KUKA KRL program: tool_gut_s.src, tool_gut_s.dat

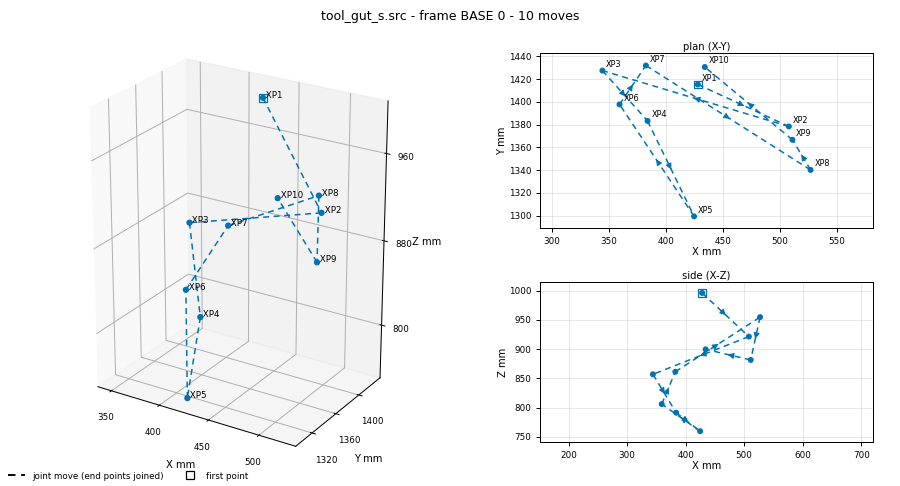
[picture p0: tool path of tool_gut_s.src in frame BASE 0, 10 of 12 moves have a stored position in this frame; points joined in program order, loops and branches not executed]
--- tool_gut_s.src ---
&ACCESS RVO
&REL 1
&PARAM EDITMASK = *
&PARAM TEMPLATE = C:\KRC\Roboter\Template\vorgabe
DEF tool_gut_s( )
;FOLD INI;%{PE}
  ;FOLD BASISTECH INI
    GLOBAL INTERRUPT DECL 3 WHEN $STOPMESS==TRUE DO IR_STOPM ( )
    INTERRUPT ON 3
    BAS (#INITMOV,0 )
  ;ENDFOLD (BASISTECH INI)
  ;FOLD USER INI
    ;Make your modifications here

  ;ENDFOLD (USER INI)
;ENDFOLD (INI)

;FOLD PTP HOME Vel=10 % DEFAULT;%{PE}%R 8.3.40,%MKUKATPBASIS,%CMOVE,%VPTP,%P 1:PTP, 2:HOME, 3:, 5:10, 7:DEFAULT
$BWDSTART=FALSE
PDAT_ACT=PDEFAULT
FDAT_ACT=FHOME
BAS(#PTP_PARAMS,10)
$H_POS=XHOME
PTP XHOME
;ENDFOLD

WAIT FOR IS_KEY_PRESSED(12)

;FOLD PTP P1 Vel=30 % PDAT1 Tool[11]:jan_ba Base[0];%{PE}%R 8.3.40,%MKUKATPBASIS,%CMOVE,%VPTP,%P 1:PTP, 2:P1, 3:, 5:30, 7:PDAT1
$BWDSTART=FALSE
PDAT_ACT=PPDAT1
FDAT_ACT=FP1
BAS(#PTP_PARAMS,30)
PTP XP1
;ENDFOLD

WAIT FOR IS_KEY_PRESSED(12)

;FOLD PTP P2 Vel=30 % PDAT2 Tool[11]:jan_ba Base[0];%{PE}%R 8.3.40,%MKUKATPBASIS,%CMOVE,%VPTP,%P 1:PTP, 2:P2, 3:, 5:30, 7:PDAT2
$BWDSTART=FALSE
PDAT_ACT=PPDAT2
FDAT_ACT=FP2
BAS(#PTP_PARAMS,30)
PTP XP2
;ENDFOLD

WAIT FOR IS_KEY_PRESSED(12)

;FOLD PTP P3 Vel=30 % PDAT3 Tool[11]:jan_ba Base[0];%{PE}%R 8.3.40,%MKUKATPBASIS,%CMOVE,%VPTP,%P 1:PTP, 2:P3, 3:, 5:30, 7:PDAT3
$BWDSTART=FALSE
PDAT_ACT=PPDAT3
FDAT_ACT=FP3
BAS(#PTP_PARAMS,30)
PTP XP3
;ENDFOLD

WAIT FOR IS_KEY_PRESSED(12)

;FOLD PTP P4 Vel=30 % PDAT4 Tool[11]:jan_ba Base[0];%{PE}%R 8.3.40,%MKUKATPBASIS,%CMOVE,%VPTP,%P 1:PTP, 2:P4, 3:, 5:30, 7:PDAT4
$BWDSTART=FALSE
PDAT_ACT=PPDAT4
FDAT_ACT=FP4
BAS(#PTP_PARAMS,30)
PTP XP4
;ENDFOLD

WAIT FOR IS_KEY_PRESSED(12)


;FOLD PTP P5 Vel=30 % PDAT5 Tool[11]:jan_ba Base[0];%{PE}%R 8.3.40,%MKUKATPBASIS,%CMOVE,%VPTP,%P 1:PTP, 2:P5, 3:, 5:30, 7:PDAT5
$BWDSTART=FALSE
PDAT_ACT=PPDAT5
FDAT_ACT=FP5
BAS(#PTP_PARAMS,30)
PTP XP5
;ENDFOLD

WAIT FOR IS_KEY_PRESSED(12)

;FOLD PTP P6 Vel=30 % PDAT6 Tool[11]:jan_ba Base[0];%{PE}%R 8.3.40,%MKUKATPBASIS,%CMOVE,%VPTP,%P 1:PTP, 2:P6, 3:, 5:30, 7:PDAT6
$BWDSTART=FALSE
PDAT_ACT=PPDAT6
FDAT_ACT=FP6
BAS(#PTP_PARAMS,30)
PTP XP6
;ENDFOLD

WAIT FOR IS_KEY_PRESSED(12)

;FOLD PTP P7 Vel=30 % PDAT7 Tool[11]:jan_ba Base[0];%{PE}%R 8.3.40,%MKUKATPBASIS,%CMOVE,%VPTP,%P 1:PTP, 2:P7, 3:, 5:30, 7:PDAT7
$BWDSTART=FALSE
PDAT_ACT=PPDAT7
FDAT_ACT=FP7
BAS(#PTP_PARAMS,30)
PTP XP7
;ENDFOLD

WAIT FOR IS_KEY_PRESSED(12)

;FOLD PTP P8 Vel=30 % PDAT8 Tool[11]:jan_ba Base[0];%{PE}%R 8.3.40,%MKUKATPBASIS,%CMOVE,%VPTP,%P 1:PTP, 2:P8, 3:, 5:30, 7:PDAT8
$BWDSTART=FALSE
PDAT_ACT=PPDAT8
FDAT_ACT=FP8
BAS(#PTP_PARAMS,30)
PTP XP8
;ENDFOLD

WAIT FOR IS_KEY_PRESSED(12)

;FOLD PTP P9 Vel=30 % PDAT9 Tool[11]:jan_ba Base[0];%{PE}%R 8.3.40,%MKUKATPBASIS,%CMOVE,%VPTP,%P 1:PTP, 2:P9, 3:, 5:30, 7:PDAT9
$BWDSTART=FALSE
PDAT_ACT=PPDAT9
FDAT_ACT=FP9
BAS(#PTP_PARAMS,30)
PTP XP9
;ENDFOLD

WAIT FOR IS_KEY_PRESSED(12)

;FOLD PTP P10 Vel=30 % PDAT10 Tool[11]:jan_ba Base[0];%{PE}%R 8.3.40,%MKUKATPBASIS,%CMOVE,%VPTP,%P 1:PTP, 2:P10, 3:, 5:30, 7:PDAT10
$BWDSTART=FALSE
PDAT_ACT=PPDAT10
FDAT_ACT=FP10
BAS(#PTP_PARAMS,30)
PTP XP10
;ENDFOLD


WAIT FOR IS_KEY_PRESSED(12)



;FOLD PTP HOME Vel=10 % DEFAULT;%{PE}%R 8.3.40,%MKUKATPBASIS,%CMOVE,%VPTP,%P 1:PTP, 2:HOME, 3:, 5:10, 7:DEFAULT
$BWDSTART=FALSE
PDAT_ACT=PDEFAULT
FDAT_ACT=FHOME
BAS(#PTP_PARAMS,10)
$H_POS=XHOME
PTP XHOME
;ENDFOLD

END

--- tool_gut_s.dat ---
&ACCESS RVO
&REL 1
&PARAM EDITMASK = *
&PARAM TEMPLATE = C:\KRC\Roboter\Template\vorgabe
DEFDAT  tool_gut_s
;FOLD EXTERNAL DECLARATIONS;%{PE}%MKUKATPBASIS,%CEXT,%VCOMMON,%P
;FOLD BASISTECH EXT;%{PE}%MKUKATPBASIS,%CEXT,%VEXT,%P
EXT  BAS (BAS_COMMAND  :IN,REAL  :IN )
DECL INT SUCCESS
;ENDFOLD (BASISTECH EXT)
;FOLD USER EXT;%{E}%MKUKATPUSER,%CEXT,%VEXT,%P
;Make your modifications here

;ENDFOLD (USER EXT)
;ENDFOLD (EXTERNAL DECLARATIONS)
DECL BASIS_SUGG_T LAST_BASIS={POINT1[] "P10                     ",POINT2[] "P10                     ",CP_PARAMS[] "CPDAT0                  ",PTP_PARAMS[] "PDAT10                  ",CONT[] "                        ",CP_VEL[] "2.0                     ",PTP_VEL[] "30                      ",SYNC_PARAMS[] "SYNCDAT                 ",SPL_NAME[] "S0                      ",A_PARAMS[] "ADAT0                   "}
DECL E6POS XP1={X 428.073151,Y 1415.33362,Z 995.893921,A 45.0438805,B 61.3839645,C -21.8034782,S 22,T 27,E1 0.00486961612,E2 20159.9980,E3 0.0,E4 0.0,E5 0.0,E6 0.0}
DECL FDAT FP1={TOOL_NO 11,BASE_NO 0,IPO_FRAME #BASE,POINT2[] " ",TQ_STATE FALSE}
DECL PDAT PPDAT1={VEL 100.000,ACC 50.0000,APO_DIST 100.000,APO_MODE #CDIS,GEAR_JERK 50.0000,EXAX_IGN 0}
DECL E6POS XP2={X 508.024689,Y 1378.40088,Z 921.330078,A -49.0426292,B 81.0973740,C -87.4984,S 22,T 27,E1 0.00486961100,E2 20159.9980,E3 0.0,E4 0.0,E5 0.0,E6 0.0}
DECL FDAT FP2={TOOL_NO 11,BASE_NO 0,IPO_FRAME #BASE,POINT2[] " ",TQ_STATE FALSE}
DECL PDAT PPDAT2={VEL 100.000,ACC 50.0000,APO_DIST 100.000,APO_MODE #CDIS,GEAR_JERK 50.0000,EXAX_IGN 0}
DECL E6POS XP3={X 344.155914,Y 1427.50085,Z 856.935913,A -65.5491104,B 67.6447372,C -167.687149,S 22,T 51,E1 0.00486961612,E2 20159.9980,E3 0.0,E4 0.0,E5 0.0,E6 0.0}
DECL FDAT FP3={TOOL_NO 11,BASE_NO 0,IPO_FRAME #BASE,POINT2[] " ",TQ_STATE FALSE}
DECL PDAT PPDAT3={VEL 100.000,ACC 50.0000,APO_DIST 100.000,APO_MODE #CDIS,GEAR_JERK 50.0000,EXAX_IGN 0}
DECL E6POS XP4={X 383.834961,Y 1383.27515,Z 791.314087,A -25.8400383,B 17.3074379,C -142.470688,S 22,T 19,E1 0.00486961612,E2 20159.9980,E3 0.0,E4 0.0,E5 0.0,E6 0.0}
DECL FDAT FP4={TOOL_NO 11,BASE_NO 0,IPO_FRAME #BASE,POINT2[] " ",TQ_STATE FALSE}
DECL PDAT PPDAT4={VEL 100.000,ACC 50.0000,APO_DIST 100.000,APO_MODE #CDIS,GEAR_JERK 50.0000,EXAX_IGN 0}
DECL E6POS XP5={X 424.737366,Y 1299.38477,Z 759.745,A -47.7535095,B -4.85419083,C -161.114349,S 18,T 3,E1 0.00486961612,E2 20159.9980,E3 0.0,E4 0.0,E5 0.0,E6 0.0}
DECL FDAT FP5={TOOL_NO 11,BASE_NO 0,IPO_FRAME #BASE,POINT2[] " ",TQ_STATE FALSE}
DECL PDAT PPDAT5={VEL 100.000,ACC 50.0000,APO_DIST 100.000,APO_MODE #CDIS,GEAR_JERK 50.0000,EXAX_IGN 0}
DECL E6POS XP6={X 359.204346,Y 1397.80554,Z 806.092102,A -4.80768585,B 12.8503466,C -133.435959,S 22,T 19,E1 0.00486961612,E2 20159.9980,E3 0.0,E4 0.0,E5 0.0,E6 0.0}
DECL FDAT FP6={TOOL_NO 11,BASE_NO 0,IPO_FRAME #BASE,POINT2[] " ",TQ_STATE FALSE}
DECL PDAT PPDAT6={VEL 100.000,ACC 50.0000,APO_DIST 100.000,APO_MODE #CDIS,GEAR_JERK 50.0000,EXAX_IGN 0}
DECL E6POS XP7={X 382.381470,Y 1431.97205,Z 861.245178,A -1.15962076,B -4.24653769,C -110.314613,S 22,T 19,E1 0.00486961612,E2 20159.9980,E3 0.0,E4 0.0,E5 0.0,E6 0.0}
DECL FDAT FP7={TOOL_NO 11,BASE_NO 0,IPO_FRAME #BASE,POINT2[] " ",TQ_STATE FALSE}
DECL PDAT PPDAT7={VEL 100.000,ACC 50.0000,APO_DIST 100.000,APO_MODE #CDIS,GEAR_JERK 50.0000,EXAX_IGN 0}
DECL E6POS XP8={X 527.139099,Y 1340.19836,Z 954.584412,A -45.5416412,B 59.4851570,C -66.5537872,S 22,T 27,E1 0.00486961612,E2 20159.9980,E3 0.0,E4 0.0,E5 0.0,E6 0.0}
DECL FDAT FP8={TOOL_NO 11,BASE_NO 0,IPO_FRAME #BASE,POINT2[] " ",TQ_STATE FALSE}
DECL PDAT PPDAT8={VEL 100.000,ACC 50.0000,APO_DIST 100.000,APO_MODE #CDIS,GEAR_JERK 50.0000,EXAX_IGN 0}
DECL E6POS XP9={X 511.166565,Y 1366.68884,Z 881.471069,A -61.5044174,B 24.6293697,C -104.485886,S 22,T 27,E1 0.00486961612,E2 20159.9980,E3 0.0,E4 0.0,E5 0.0,E6 0.0}
DECL FDAT FP9={TOOL_NO 11,BASE_NO 0,IPO_FRAME #BASE,POINT2[] " ",TQ_STATE FALSE}
DECL PDAT PPDAT9={VEL 100.000,ACC 50.0000,APO_DIST 100.000,APO_MODE #CDIS,GEAR_JERK 50.0000,EXAX_IGN 0}
DECL E6POS XP10={X 434.148468,Y 1430.66406,Z 899.584106,A -17.7071095,B -22.2916451,C -97.5115356,S 22,T 27,E1 0.00486961612,E2 20159.9980,E3 0.0,E4 0.0,E5 0.0,E6 0.0}
DECL FDAT FP10={TOOL_NO 11,BASE_NO 0,IPO_FRAME #BASE,POINT2[] " ",TQ_STATE FALSE}
DECL PDAT PPDAT10={VEL 100.000,ACC 50.0000,APO_DIST 100.000,APO_MODE #CDIS,GEAR_JERK 50.0000,EXAX_IGN 0}
ENDDAT
